// TIA Portal project "3_Fazlı_Asenkron_Motora_Direkt_Yol_Verme" (V15)

(* hardware
DEVICE "S7-1200 station_1"  S7-1200 Station
   slot 0: "Rack_0"  S7-1200 Rack  Rack  V1.0
   slot 1: "PLC_1"  CPU 1212C DC/DC/DC  6ES7 212-1AE40-0XB0  V4.2
*)

// ===== PLC "PLC_1"  CPU 1212C DC/DC/DC =====

VAR_GLOBAL   // PLC tag table "Default tag table"
   "I_THERMAL_RELAY" AT %I0.0 : Bool;
   "I_STOP_BTN" AT %I0.1 : Bool;
   "I_START_BTN" AT %I0.2 : Bool;
   "Q_MOTOR" AT %Q0.0 : Bool;
END_VAR

ORGANIZATION_BLOCK "Main"   // OB1, LAD, ProgramCycle
TITLE = "Main Program Sweep (Cycle)"
{ S7_Optimized_Access := 'TRUE' }
VERSION : 0.1
   VAR_INPUT
      Initial_Call : Bool;   // Initial call of this OB
      Remanence : Bool;   // =True, if remanent data are available
   END_VAR
BEGIN

REGION Network 1
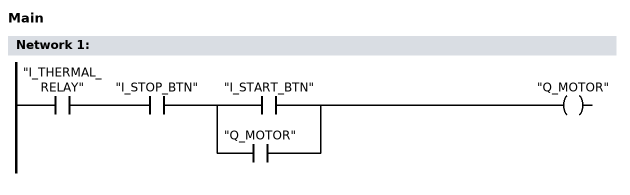
   RUNG wire#powerrail
      Contact( "I_THERMAL_RELAY" )
      Contact( "I_STOP_BTN" )
      wire#w1
      Contact( "I_START_BTN" )
      wire#w2
      Coil( "Q_MOTOR" )
   END_RUNG
   RUNG wire#w1
      Contact( "Q_MOTOR" )
   END_RUNG wire#w2
   // the same network as SCL:
   "Q_MOTOR" := "I_THERMAL_RELAY" AND "I_STOP_BTN" AND ("I_START_BTN" OR "Q_MOTOR");
END_REGION
END_ORGANIZATION_BLOCK